(* PLC project Senza_nome, Sconosciuto Senza_nome 1 *)
(* stored: creationDateTime 2026-08-25T11:39:47, modificationDateTime 2026-08-25T11:46:19 *)

PROGRAM program0
  VAR
    SR0 : SR;
    SR1 : SR;
    S1 : BOOL;
    S2 : BOOL;
    RESET : BOOL;
    LED1 : BOOL;
    LED2 : BOOL;
  END_VAR

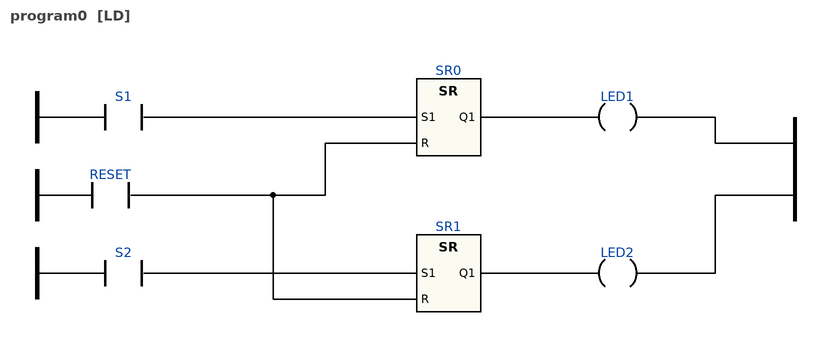
(* LD diagram, written out as Structured Text *)
SR0(S1 := S1, R := RESET);
LED1 := SR0.Q1;
SR1(S1 := S2, R := RESET);
LED2 := SR1.Q1;
END_PROGRAM

CONFIGURATION Config0
  RESOURCE Res0 ON PLC
    TASK task0(INTERVAL := T#20ms, PRIORITY := 0);
    PROGRAM instance0 WITH task0 : program0;
  END_RESOURCE
END_CONFIGURATION
